# EPICS autosave request: arrowApp/Db/NDPluginArrow_settings.req
# Nothing extra needed beyond NDPluginBase_settings.req for now
file "NDPluginBase_settings.req", P=$(P), R=$(R)
file "NDFile_settings.req", P=$(P), R=$(R)
